// This function has been automatically generated from the project information.
VAR_GLOBAL CONSTANT
	{attribute 'const_non_replaced'}
	stLibVersion_Base_Elements : ST_LibVersion := (iMajor := 0, iMinor := 0, iBuild := 1, iRevision := 65, sVersion := '0.0.1.65');
END_VAR

(* stored: Version 1.1.0.1, ProductVersion 3.1.0.36
   GVL Global_Version: Id {6b6dc6af-b87e-41c1-b05f-94651408b334} *)
